% RSLogix 500 project Automated Water Storage & Filtration Control System.RSS, saved by version 8.30.00.16 %
PROJECT "UNTITLED"    % processor: Bul.1763 MicroLogix 1100 Series B %

PROGRAM FILES
  LAD 2 "MAIN"  9 rungs
  LAD 3 "IO"  13 rungs
  LAD 4 "HOA"  36 rungs
  LAD 5 "CONTROLS"  16 rungs
  LAD 6 "RUNTIME"  6 rungs
  LAD 7 "BACKWASH"  16 rungs
  LAD 8 "ALARM"  17 rungs
  LAD 9 "SIMULATION"  9 rungs  % SIMULATED IO %
  LAD 10 "SETTOAUTO"  3 rungs

DATA FILES
  O0 OUTPUT  4 elements
  I1 INPUT  13 elements
  S2 STATUS  66 elements
  B3 BINARY  9 elements
  T4 TIMER  11 elements
  C5 COUNTER  1 elements
  R6 CONTROL  1 elements
  N7 INTEGER  19 elements
  F8 FLOAT  15 elements

LADDER 2 "MAIN"
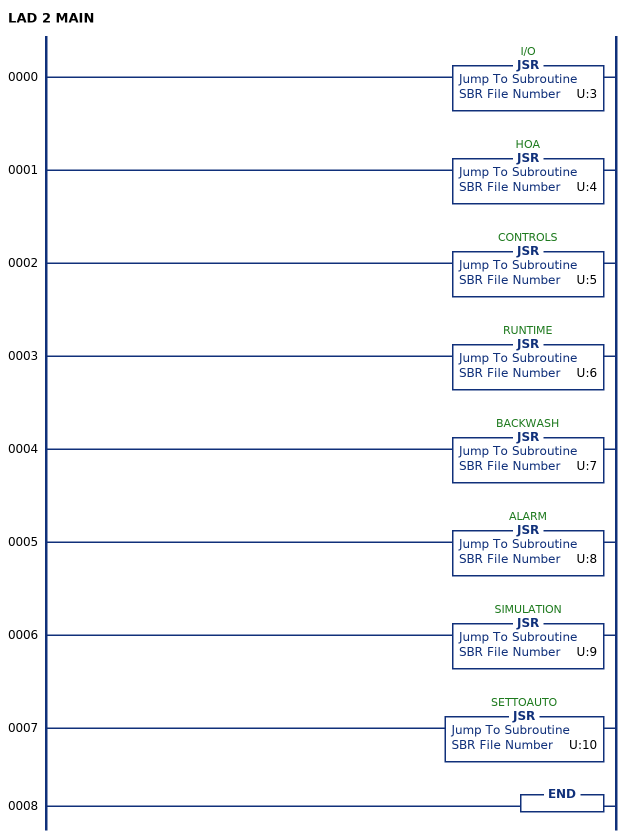
% Rung: 0 %
SOR JSR U:3 EOR
%   U:3  "I/O" %
% Rung: 1 %
SOR JSR U:4 EOR
%   U:4  "HOA" %
% Rung: 2 %
SOR JSR U:5 EOR
%   U:5  "CONTROLS" %
% Rung: 3 %
SOR JSR U:6 EOR
%   U:6  "RUNTIME" %
% Rung: 4 %
SOR JSR U:7 EOR
%   U:7  "BACKWASH" %
% Rung: 5 %
SOR JSR U:8 EOR
%   U:8  "ALARM" %
% Rung: 6 %
SOR JSR U:9 EOR
%   U:9  "SIMULATION" %
% Rung: 7 %
SOR JSR U:10 EOR
%   U:10  "SETTOAUTO" %
% Rung: 8 %
SOR END EOR

LADDER 3 "IO"
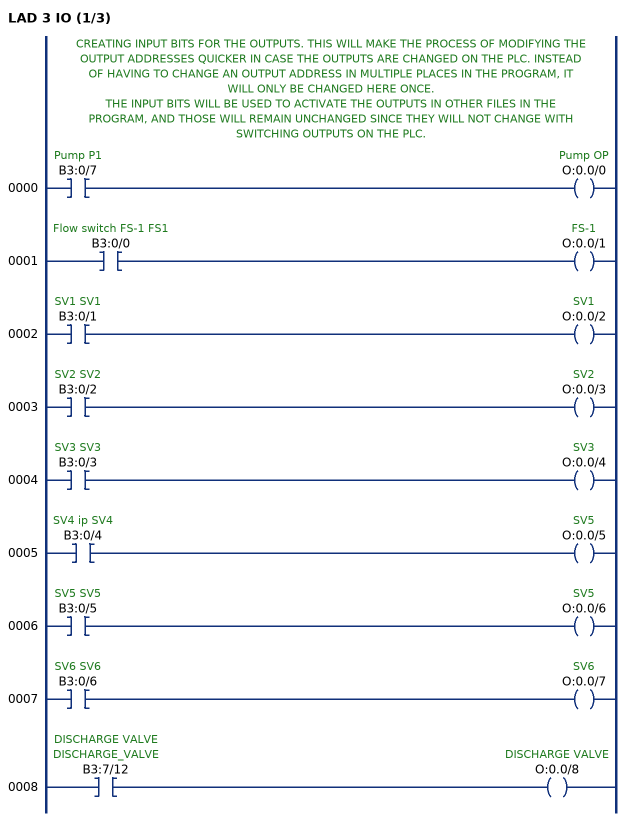
% Rung: 0 %
% CREATING INPUT BITS FOR THE OUTPUTS. THIS WILL MAKE THE PROCESS OF MODIFYING THE OUTPUT ADDRESSES QUICKER IN CASE THE OUTPUTS ARE CHANGED ON THE PLC. INSTEAD OF HAVING TO CHANGE AN OUTPUT ADDRESS IN MULTIPLE PLACES IN THE PROGRAM, IT WILL ONLY BE CHANGED HERE ONCE.
% THE INPUT BITS WILL BE USED TO ACTIVATE THE OUTPUTS IN OTHER FILES IN THE PROGRAM, AND THOSE WILL REMAIN UNCHANGED SINCE THEY WILL NOT CHANGE WITH SWITCHING OUTPUTS ON THE PLC. %
SOR XIC B3:0/7 OTE O:0.0/0 EOR
%   B3:0/7  P1  "Pump" %
%   O:0.0/0  "Pump OP" %
% Rung: 1 %
SOR XIC B3:0/0 OTE O:0.0/1 EOR
%   B3:0/0  FS1  "Flow switch FS-1" %
%   O:0.0/1  "FS-1" %
% Rung: 2 %
SOR XIC B3:0/1 OTE O:0.0/2 EOR
%   B3:0/1  SV1  "SV1" %
%   O:0.0/2  "SV1" %
% Rung: 3 %
SOR XIC B3:0/2 OTE O:0.0/3 EOR
%   B3:0/2  SV2  "SV2" %
%   O:0.0/3  "SV2" %
% Rung: 4 %
SOR XIC B3:0/3 OTE O:0.0/4 EOR
%   B3:0/3  SV3  "SV3" %
%   O:0.0/4  "SV3" %
% Rung: 5 %
SOR XIC B3:0/4 OTE O:0.0/5 EOR
%   B3:0/4  SV4  "SV4 ip" %
%   O:0.0/5  "SV5" %
% Rung: 6 %
SOR XIC B3:0/5 OTE O:0.0/6 EOR
%   B3:0/5  SV5  "SV5" %
%   O:0.0/6  "SV5" %
% Rung: 7 %
SOR XIC B3:0/6 OTE O:0.0/7 EOR
%   B3:0/6  SV6  "SV6" %
%   O:0.0/7  "SV6" %
% Rung: 8 %
SOR XIC B3:7/12 OTE O:0.0/8 EOR
%   B3:7/12  DISCHARGE_VALVE  "DISCHARGE VALVE" %
%   O:0.0/8  "DISCHARGE VALVE" %

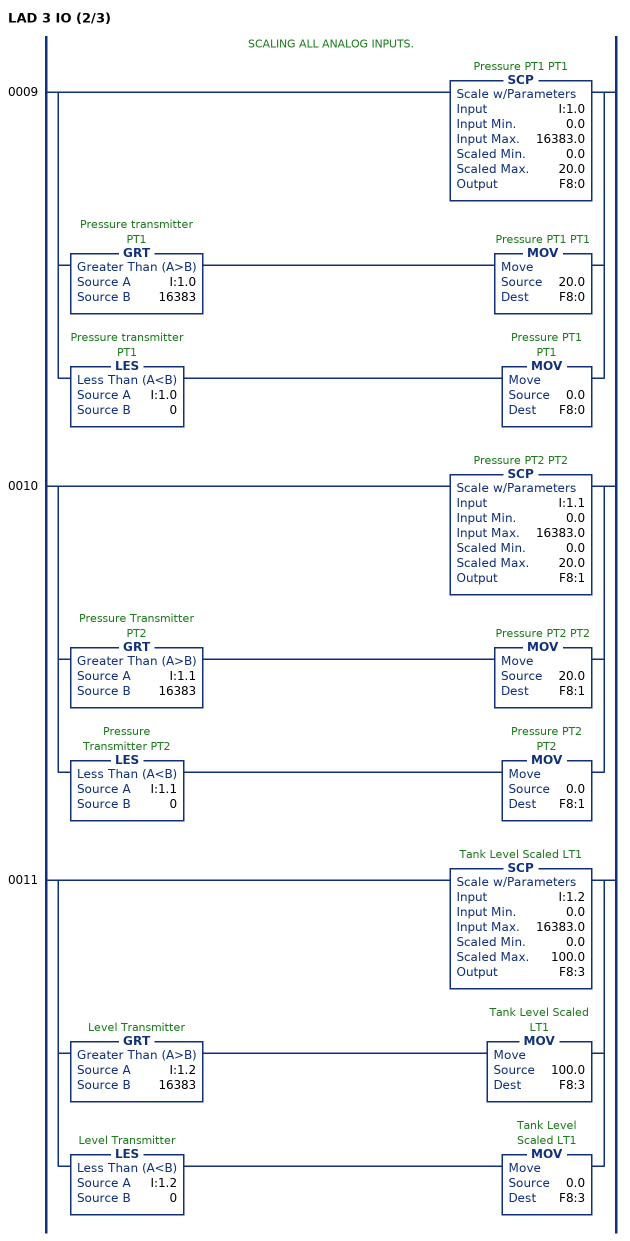
% Rung: 9 %
% SCALING ALL ANALOG INPUTS. %
SOR BST SCP I:1.0 0.0 16383.0 0.0 20.0 F8:0 NXB GRT I:1.0 16383 MOV 20.0 F8:0 NXB LES I:1.0 0 MOV 0.0 F8:0 BND EOR
%   I:1.0  "Pressure transmitter PT1" %
%   F8:0  PT1  "Pressure PT1" %
% Rung: 10 %
SOR BST SCP I:1.1 0.0 16383.0 0.0 20.0 F8:1 NXB GRT I:1.1 16383 MOV 20.0 F8:1 NXB LES I:1.1 0 MOV 0.0 F8:1 BND EOR
%   I:1.1  "Pressure Transmitter PT2" %
%   F8:1  PT2  "Pressure PT2" %
% Rung: 11 %
SOR BST SCP I:1.2 0.0 16383.0 0.0 100.0 F8:3 NXB GRT I:1.2 16383 MOV 100.0 F8:3 NXB LES I:1.2 0 MOV 0.0 F8:3 BND EOR
%   I:1.2  "Level Transmitter" %
%   F8:3  LT1  "Tank Level Scaled" %

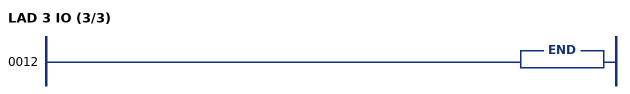
% Rung: 12 %
SOR END EOR

LADDER 4 "HOA"
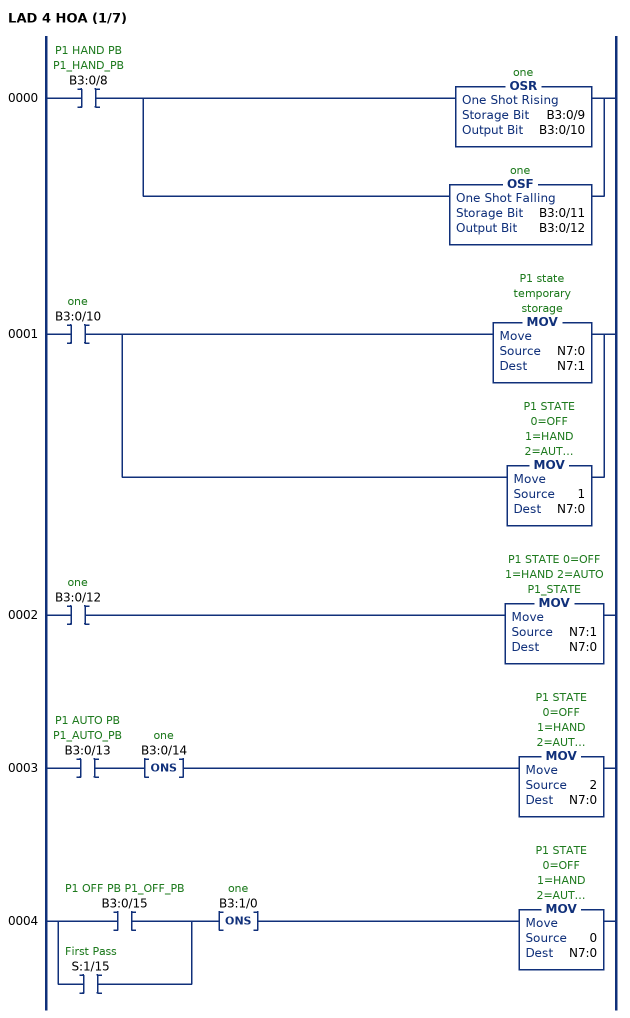
% Rung: 0 %
SOR XIC B3:0/8 BST OSR B3:0/9 B3:0/10 NXB OSF B3:0/11 B3:0/12 BND EOR
%   B3:0/8  P1_HAND_PB  "P1 HAND PB" %
%   B3:0/9  "one" %
%   B3:0/10  "one" %
%   B3:0/11  "one" %
%   B3:0/12  "one" %
% Rung: 1 %
SOR XIC B3:0/10 BST MOV N7:0 N7:1 NXB MOV 1 N7:0 BND EOR
%   B3:0/10  "one" %
%   N7:0  P1_STATE  "P1 STATE 0=OFF 1=HAND 2=AUTO" %
%   N7:1  "P1 state temporary storage" %
% Rung: 2 %
SOR XIC B3:0/12 MOV N7:1 N7:0 EOR
%   B3:0/12  "one" %
%   N7:1  "P1 state temporary storage" %
%   N7:0  P1_STATE  "P1 STATE 0=OFF 1=HAND 2=AUTO" %
% Rung: 3 %
SOR XIC B3:0/13 ONS B3:0/14 MOV 2 N7:0 EOR
%   B3:0/13  P1_AUTO_PB  "P1 AUTO PB" %
%   B3:0/14  "one" %
%   N7:0  P1_STATE  "P1 STATE 0=OFF 1=HAND 2=AUTO" %
% Rung: 4 %
SOR BST XIC B3:0/15 NXB XIC S:1/15 BND ONS B3:1/0 MOV 0 N7:0 EOR
%   B3:0/15  P1_OFF_PB  "P1 OFF PB" %
%   S:1/15  "First Pass" %
%   B3:1/0  "one" %
%   N7:0  P1_STATE  "P1 STATE 0=OFF 1=HAND 2=AUTO" %

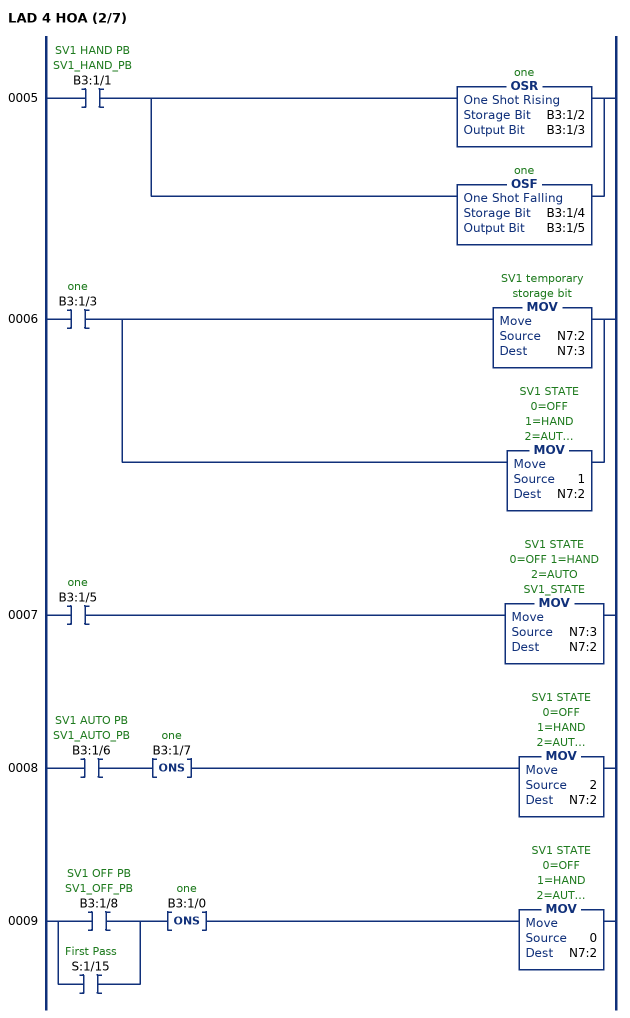
% Rung: 5 %
SOR XIC B3:1/1 BST OSR B3:1/2 B3:1/3 NXB OSF B3:1/4 B3:1/5 BND EOR
%   B3:1/1  SV1_HAND_PB  "SV1 HAND PB" %
%   B3:1/2  "one" %
%   B3:1/3  "one" %
%   B3:1/4  "one" %
%   B3:1/5  "one" %
% Rung: 6 %
SOR XIC B3:1/3 BST MOV N7:2 N7:3 NXB MOV 1 N7:2 BND EOR
%   B3:1/3  "one" %
%   N7:2  SV1_STATE  "SV1 STATE 0=OFF 1=HAND 2=AUTO" %
%   N7:3  "SV1 temporary storage bit" %
% Rung: 7 %
SOR XIC B3:1/5 MOV N7:3 N7:2 EOR
%   B3:1/5  "one" %
%   N7:3  "SV1 temporary storage bit" %
%   N7:2  SV1_STATE  "SV1 STATE 0=OFF 1=HAND 2=AUTO" %
% Rung: 8 %
SOR XIC B3:1/6 ONS B3:1/7 MOV 2 N7:2 EOR
%   B3:1/6  SV1_AUTO_PB  "SV1 AUTO PB" %
%   B3:1/7  "one" %
%   N7:2  SV1_STATE  "SV1 STATE 0=OFF 1=HAND 2=AUTO" %
% Rung: 9 %
SOR BST XIC B3:1/8 NXB XIC S:1/15 BND ONS B3:1/0 MOV 0 N7:2 EOR
%   B3:1/8  SV1_OFF_PB  "SV1 OFF PB" %
%   S:1/15  "First Pass" %
%   B3:1/0  "one" %
%   N7:2  SV1_STATE  "SV1 STATE 0=OFF 1=HAND 2=AUTO" %

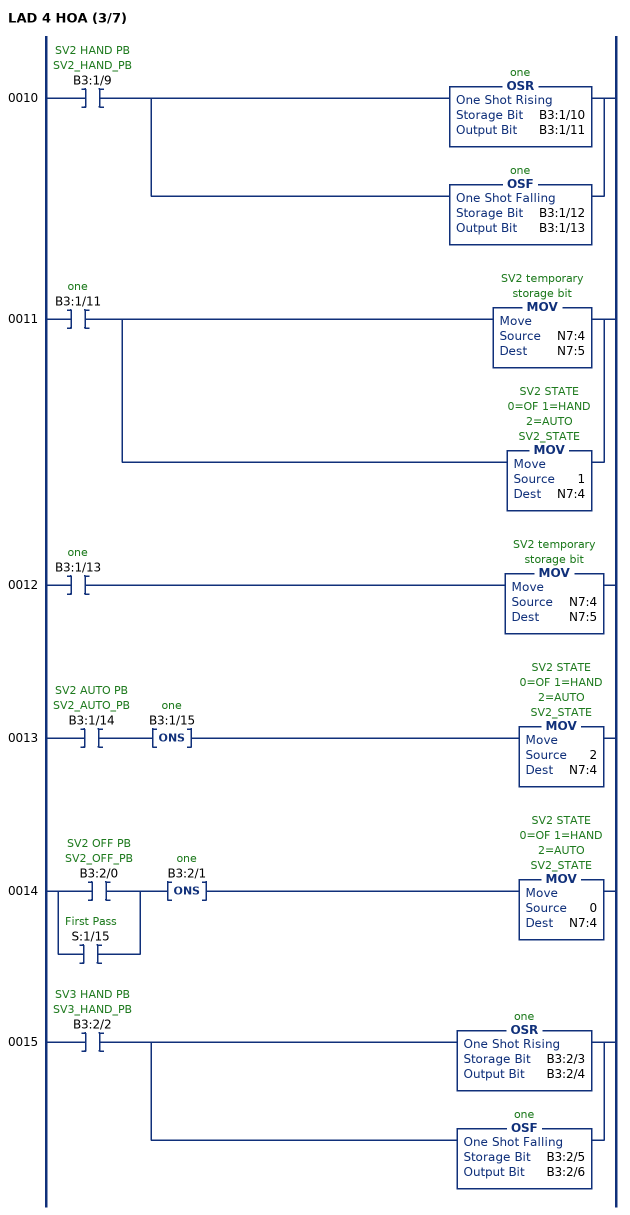
% Rung: 10 %
SOR XIC B3:1/9 BST OSR B3:1/10 B3:1/11 NXB OSF B3:1/12 B3:1/13 BND EOR
%   B3:1/9  SV2_HAND_PB  "SV2 HAND PB" %
%   B3:1/10  "one" %
%   B3:1/11  "one" %
%   B3:1/12  "one" %
%   B3:1/13  "one" %
% Rung: 11 %
SOR XIC B3:1/11 BST MOV N7:4 N7:5 NXB MOV 1 N7:4 BND EOR
%   B3:1/11  "one" %
%   N7:4  SV2_STATE  "SV2 STATE 0=OF 1=HAND 2=AUTO" %
%   N7:5  "SV2 temporary storage bit" %
% Rung: 12 %
SOR XIC B3:1/13 MOV N7:4 N7:5 EOR
%   B3:1/13  "one" %
%   N7:4  SV2_STATE  "SV2 STATE 0=OF 1=HAND 2=AUTO" %
%   N7:5  "SV2 temporary storage bit" %
% Rung: 13 %
SOR XIC B3:1/14 ONS B3:1/15 MOV 2 N7:4 EOR
%   B3:1/14  SV2_AUTO_PB  "SV2 AUTO PB" %
%   B3:1/15  "one" %
%   N7:4  SV2_STATE  "SV2 STATE 0=OF 1=HAND 2=AUTO" %
% Rung: 14 %
SOR BST XIC B3:2/0 NXB XIC S:1/15 BND ONS B3:2/1 MOV 0 N7:4 EOR
%   B3:2/0  SV2_OFF_PB  "SV2 OFF PB" %
%   S:1/15  "First Pass" %
%   B3:2/1  "one" %
%   N7:4  SV2_STATE  "SV2 STATE 0=OF 1=HAND 2=AUTO" %
% Rung: 15 %
SOR XIC B3:2/2 BST OSR B3:2/3 B3:2/4 NXB OSF B3:2/5 B3:2/6 BND EOR
%   B3:2/2  SV3_HAND_PB  "SV3 HAND PB" %
%   B3:2/3  "one" %
%   B3:2/4  "one" %
%   B3:2/5  "one" %
%   B3:2/6  "one" %

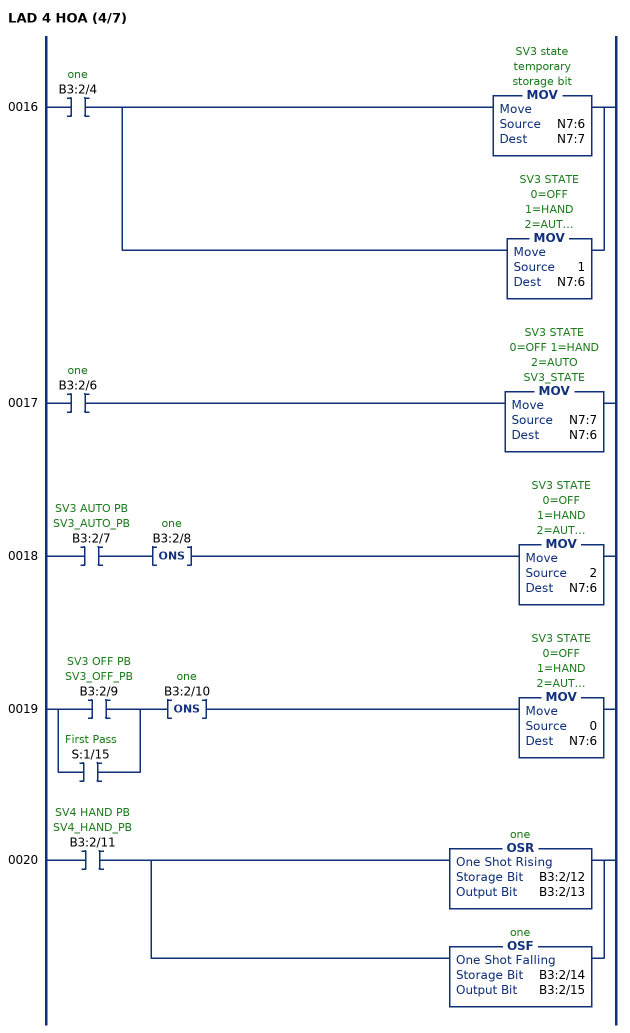
% Rung: 16 %
SOR XIC B3:2/4 BST MOV N7:6 N7:7 NXB MOV 1 N7:6 BND EOR
%   B3:2/4  "one" %
%   N7:6  SV3_STATE  "SV3 STATE 0=OFF 1=HAND 2=AUTO" %
%   N7:7  "SV3 state temporary storage bit" %
% Rung: 17 %
SOR XIC B3:2/6 MOV N7:7 N7:6 EOR
%   B3:2/6  "one" %
%   N7:7  "SV3 state temporary storage bit" %
%   N7:6  SV3_STATE  "SV3 STATE 0=OFF 1=HAND 2=AUTO" %
% Rung: 18 %
SOR XIC B3:2/7 ONS B3:2/8 MOV 2 N7:6 EOR
%   B3:2/7  SV3_AUTO_PB  "SV3 AUTO PB" %
%   B3:2/8  "one" %
%   N7:6  SV3_STATE  "SV3 STATE 0=OFF 1=HAND 2=AUTO" %
% Rung: 19 %
SOR BST XIC B3:2/9 NXB XIC S:1/15 BND ONS B3:2/10 MOV 0 N7:6 EOR
%   B3:2/9  SV3_OFF_PB  "SV3 OFF PB" %
%   S:1/15  "First Pass" %
%   B3:2/10  "one" %
%   N7:6  SV3_STATE  "SV3 STATE 0=OFF 1=HAND 2=AUTO" %
% Rung: 20 %
SOR XIC B3:2/11 BST OSR B3:2/12 B3:2/13 NXB OSF B3:2/14 B3:2/15 BND EOR
%   B3:2/11  SV4_HAND_PB  "SV4 HAND PB" %
%   B3:2/12  "one" %
%   B3:2/13  "one" %
%   B3:2/14  "one" %
%   B3:2/15  "one" %

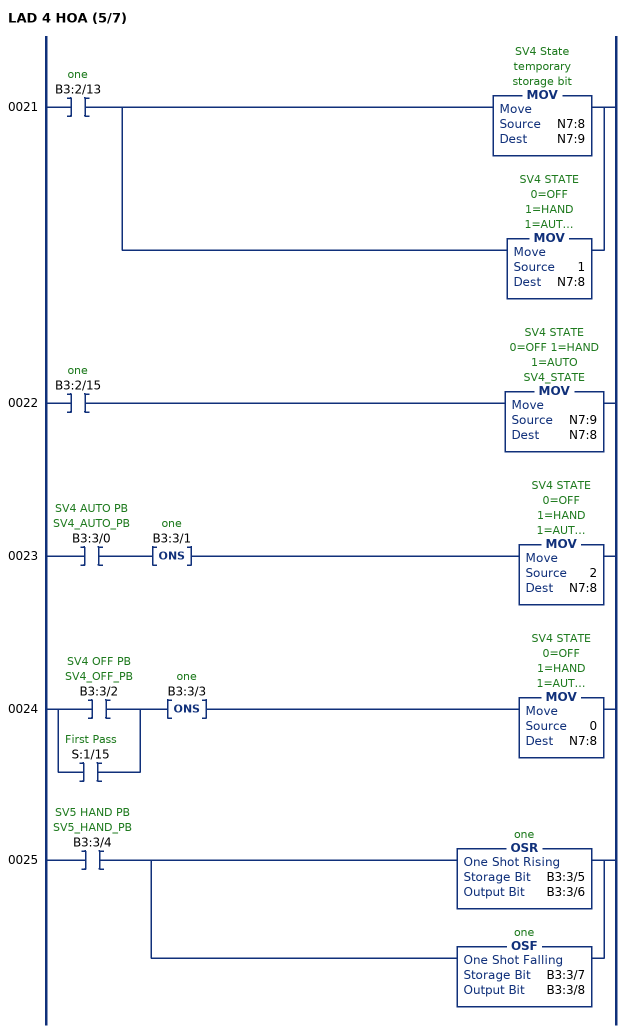
% Rung: 21 %
SOR XIC B3:2/13 BST MOV N7:8 N7:9 NXB MOV 1 N7:8 BND EOR
%   B3:2/13  "one" %
%   N7:8  SV4_STATE  "SV4 STATE 0=OFF 1=HAND 1=AUTO" %
%   N7:9  "SV4 State temporary storage bit" %
% Rung: 22 %
SOR XIC B3:2/15 MOV N7:9 N7:8 EOR
%   B3:2/15  "one" %
%   N7:9  "SV4 State temporary storage bit" %
%   N7:8  SV4_STATE  "SV4 STATE 0=OFF 1=HAND 1=AUTO" %
% Rung: 23 %
SOR XIC B3:3/0 ONS B3:3/1 MOV 2 N7:8 EOR
%   B3:3/0  SV4_AUTO_PB  "SV4 AUTO PB" %
%   B3:3/1  "one" %
%   N7:8  SV4_STATE  "SV4 STATE 0=OFF 1=HAND 1=AUTO" %
% Rung: 24 %
SOR BST XIC B3:3/2 NXB XIC S:1/15 BND ONS B3:3/3 MOV 0 N7:8 EOR
%   B3:3/2  SV4_OFF_PB  "SV4 OFF PB" %
%   S:1/15  "First Pass" %
%   B3:3/3  "one" %
%   N7:8  SV4_STATE  "SV4 STATE 0=OFF 1=HAND 1=AUTO" %
% Rung: 25 %
SOR XIC B3:3/4 BST OSR B3:3/5 B3:3/6 NXB OSF B3:3/7 B3:3/8 BND EOR
%   B3:3/4  SV5_HAND_PB  "SV5 HAND PB" %
%   B3:3/5  "one" %
%   B3:3/6  "one" %
%   B3:3/7  "one" %
%   B3:3/8  "one" %

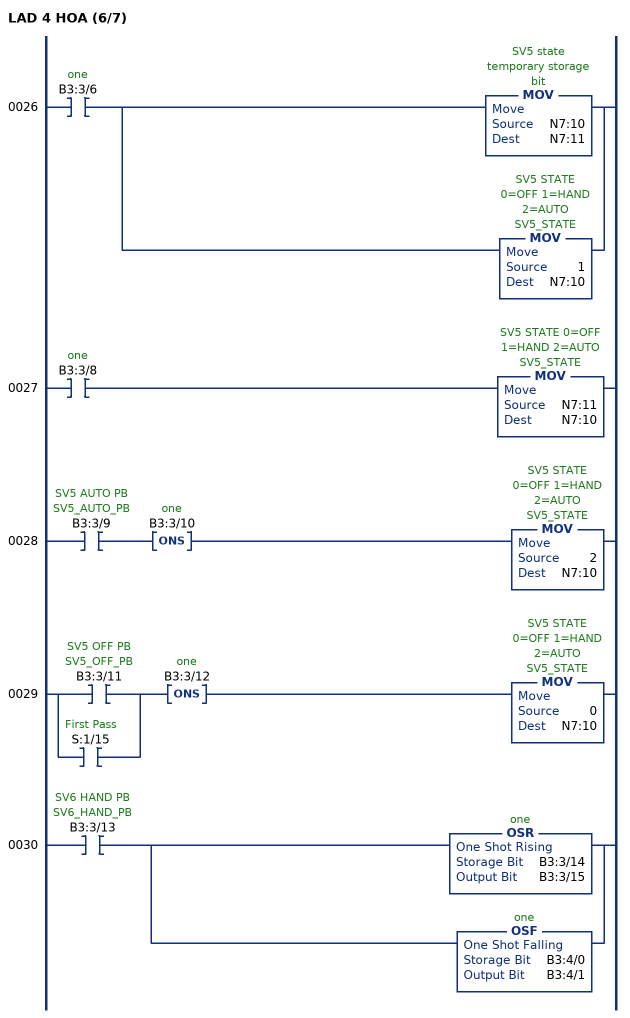
% Rung: 26 %
SOR XIC B3:3/6 BST MOV N7:10 N7:11 NXB MOV 1 N7:10 BND EOR
%   B3:3/6  "one" %
%   N7:10  SV5_STATE  "SV5 STATE 0=OFF 1=HAND 2=AUTO" %
%   N7:11  "SV5 state temporary storage bit" %
% Rung: 27 %
SOR XIC B3:3/8 MOV N7:11 N7:10 EOR
%   B3:3/8  "one" %
%   N7:11  "SV5 state temporary storage bit" %
%   N7:10  SV5_STATE  "SV5 STATE 0=OFF 1=HAND 2=AUTO" %
% Rung: 28 %
SOR XIC B3:3/9 ONS B3:3/10 MOV 2 N7:10 EOR
%   B3:3/9  SV5_AUTO_PB  "SV5 AUTO PB" %
%   B3:3/10  "one" %
%   N7:10  SV5_STATE  "SV5 STATE 0=OFF 1=HAND 2=AUTO" %
% Rung: 29 %
SOR BST XIC B3:3/11 NXB XIC S:1/15 BND ONS B3:3/12 MOV 0 N7:10 EOR
%   B3:3/11  SV5_OFF_PB  "SV5 OFF PB" %
%   S:1/15  "First Pass" %
%   B3:3/12  "one" %
%   N7:10  SV5_STATE  "SV5 STATE 0=OFF 1=HAND 2=AUTO" %
% Rung: 30 %
SOR XIC B3:3/13 BST OSR B3:3/14 B3:3/15 NXB OSF B3:4/0 B3:4/1 BND EOR
%   B3:3/13  SV6_HAND_PB  "SV6 HAND PB" %
%   B3:3/14  "one" %
%   B3:3/15  "one" %
%   B3:4/0  "one" %
%   B3:4/1  "one" %

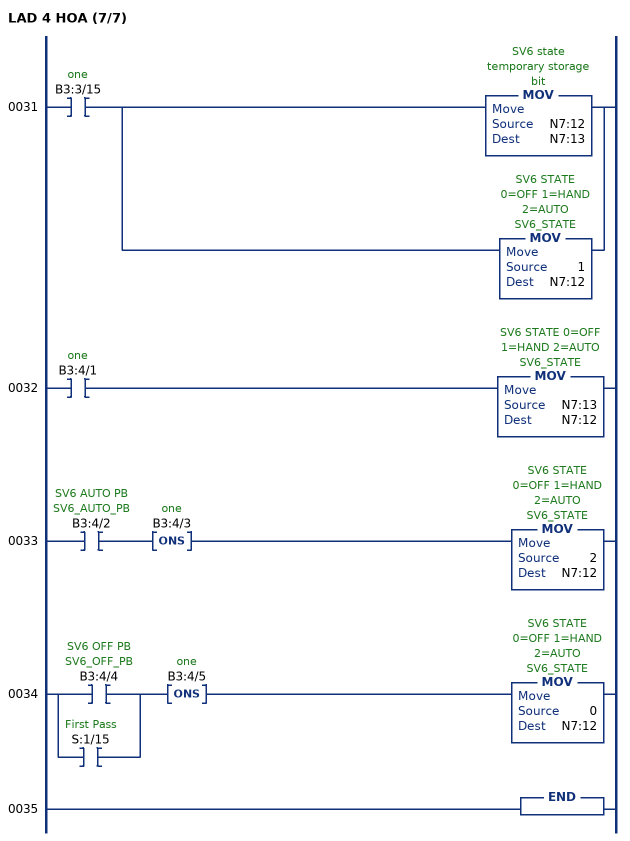
% Rung: 31 %
SOR XIC B3:3/15 BST MOV N7:12 N7:13 NXB MOV 1 N7:12 BND EOR
%   B3:3/15  "one" %
%   N7:12  SV6_STATE  "SV6 STATE 0=OFF 1=HAND 2=AUTO" %
%   N7:13  "SV6 state temporary storage bit" %
% Rung: 32 %
SOR XIC B3:4/1 MOV N7:13 N7:12 EOR
%   B3:4/1  "one" %
%   N7:13  "SV6 state temporary storage bit" %
%   N7:12  SV6_STATE  "SV6 STATE 0=OFF 1=HAND 2=AUTO" %
% Rung: 33 %
SOR XIC B3:4/2 ONS B3:4/3 MOV 2 N7:12 EOR
%   B3:4/2  SV6_AUTO_PB  "SV6 AUTO PB" %
%   B3:4/3  "one" %
%   N7:12  SV6_STATE  "SV6 STATE 0=OFF 1=HAND 2=AUTO" %
% Rung: 34 %
SOR BST XIC B3:4/4 NXB XIC S:1/15 BND ONS B3:4/5 MOV 0 N7:12 EOR
%   B3:4/4  SV6_OFF_PB  "SV6 OFF PB" %
%   S:1/15  "First Pass" %
%   B3:4/5  "one" %
%   N7:12  SV6_STATE  "SV6 STATE 0=OFF 1=HAND 2=AUTO" %
% Rung: 35 %
SOR END EOR

LADDER 5 "CONTROLS"
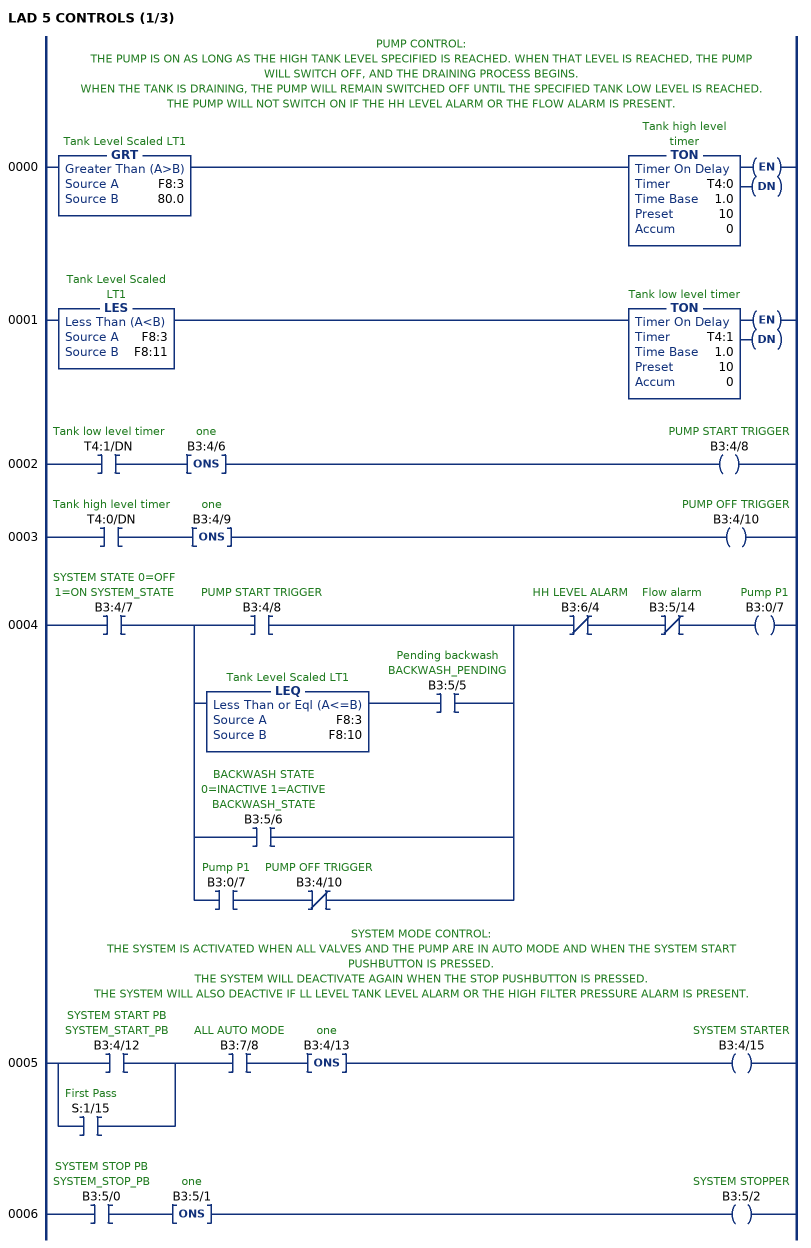
% Rung: 0 %
% PUMP CONTROL:
% THE PUMP IS ON AS LONG AS THE HIGH TANK LEVEL SPECIFIED IS REACHED. WHEN THAT LEVEL IS REACHED, THE PUMP WILL SWITCH OFF, AND THE DRAINING PROCESS BEGINS.
% WHEN THE TANK IS DRAINING, THE PUMP WILL REMAIN SWITCHED OFF UNTIL THE SPECIFIED TANK LOW LEVEL IS REACHED.
% THE PUMP WILL NOT SWITCH ON IF THE HH LEVEL ALARM OR THE FLOW ALARM IS PRESENT. %
SOR GRT F8:3 80.0 TON T4:0 1.0 10 0 EOR
%   F8:3  LT1  "Tank Level Scaled" %
%   T4:0  "Tank high level timer" %
% Rung: 1 %
SOR LES F8:3 F8:11 TON T4:1 1.0 10 0 EOR
%   F8:3  LT1  "Tank Level Scaled" %
%   F8:11  L_LEVEL  "L_TANK_LEVEL" %
%   T4:1  "Tank low level timer" %
% Rung: 2 %
SOR XIC T4:1/DN ONS B3:4/6 OTE B3:4/8 EOR
%   T4:1  "Tank low level timer" %
%   B3:4/6  "one" %
%   B3:4/8  "PUMP START TRIGGER" %
% Rung: 3 %
SOR XIC T4:0/DN ONS B3:4/9 OTE B3:4/10 EOR
%   T4:0  "Tank high level timer" %
%   B3:4/9  "one" %
%   B3:4/10  "PUMP OFF TRIGGER" %
% Rung: 4 %
SOR XIC B3:4/7 BST XIC B3:4/8 NXB LEQ F8:3 F8:10 XIC B3:5/5 NXB XIC B3:5/6 NXB XIC B3:0/7 XIO B3:4/10 BND XIO B3:6/4 XIO B3:5/14 OTE B3:0/7 EOR
%   B3:4/7  SYSTEM_STATE  "SYSTEM STATE 0=OFF 1=ON" %
%   B3:4/8  "PUMP START TRIGGER" %
%   F8:3  LT1  "Tank Level Scaled" %
%   F8:10  H_LEVEL  "H_TANK_LEVEL" %
%   B3:5/5  BACKWASH_PENDING  "Pending backwash" %
%   B3:5/6  BACKWASH_STATE  "BACKWASH STATE 0=INACTIVE 1=ACTIVE" %
%   B3:0/7  P1  "Pump" %
%   B3:4/10  "PUMP OFF TRIGGER" %
%   B3:6/4  "HH LEVEL ALARM" %
%   B3:5/14  "Flow alarm" %
% Rung: 5 %
% SYSTEM MODE CONTROL:
% THE SYSTEM IS ACTIVATED WHEN ALL VALVES AND THE PUMP ARE IN AUTO MODE AND WHEN THE SYSTEM START PUSHBUTTON IS PRESSED.
% THE SYSTEM WILL DEACTIVATE AGAIN WHEN THE STOP PUSHBUTTON IS PRESSED.
% THE SYSTEM WILL ALSO DEACTIVE IF LL LEVEL TANK LEVEL ALARM OR THE HIGH FILTER PRESSURE ALARM IS PRESENT. %
SOR BST XIC B3:4/12 NXB XIC S:1/15 BND XIC B3:7/8 ONS B3:4/13 OTE B3:4/15 EOR
%   B3:4/12  SYSTEM_START_PB  "SYSTEM START PB" %
%   S:1/15  "First Pass" %
%   B3:7/8  "ALL AUTO MODE" %
%   B3:4/13  "one" %
%   B3:4/15  "SYSTEM STARTER" %
% Rung: 6 %
SOR XIC B3:5/0 ONS B3:5/1 OTE B3:5/2 EOR
%   B3:5/0  SYSTEM_STOP_PB  "SYSTEM STOP PB" %
%   B3:5/1  "one" %
%   B3:5/2  "SYSTEM STOPPER" %

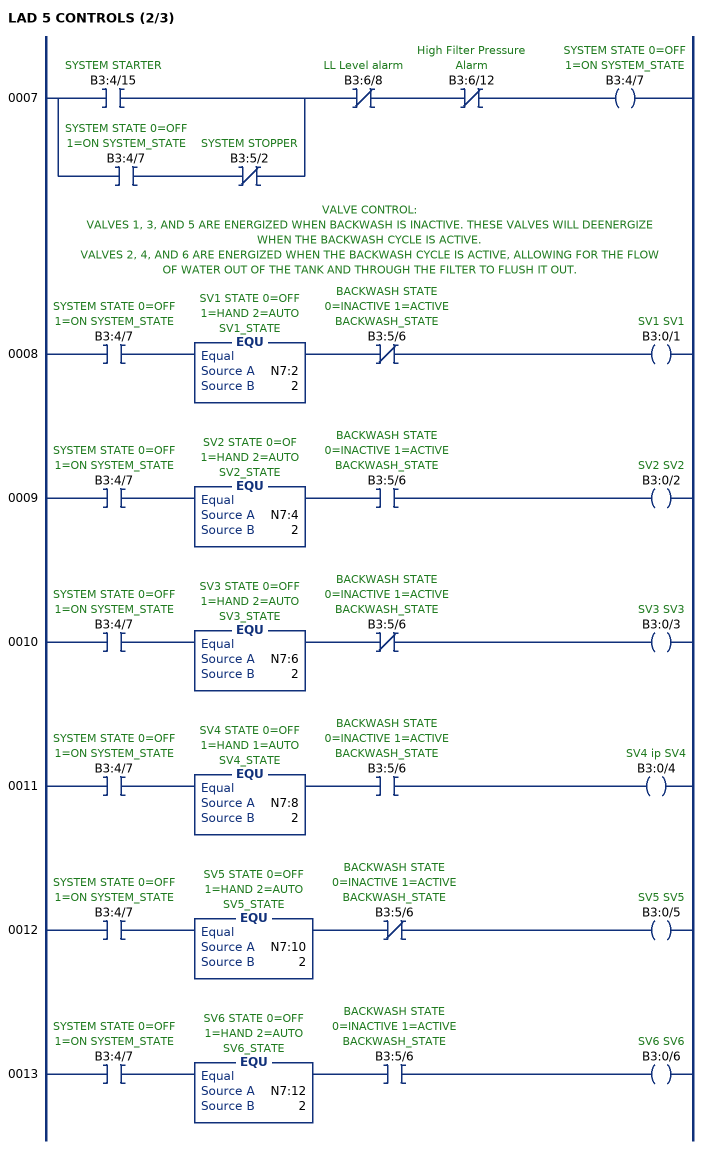
% Rung: 7 %
SOR BST XIC B3:4/15 NXB XIC B3:4/7 XIO B3:5/2 BND XIO B3:6/8 XIO B3:6/12 OTE B3:4/7 EOR
%   B3:4/15  "SYSTEM STARTER" %
%   B3:4/7  SYSTEM_STATE  "SYSTEM STATE 0=OFF 1=ON" %
%   B3:5/2  "SYSTEM STOPPER" %
%   B3:6/8  "LL Level alarm" %
%   B3:6/12  "High Filter Pressure Alarm" %
% Rung: 8 %
% VALVE CONTROL:
% VALVES 1, 3, AND 5 ARE ENERGIZED WHEN BACKWASH IS INACTIVE. THESE VALVES WILL DEENERGIZE WHEN THE BACKWASH CYCLE IS ACTIVE.
% VALVES 2, 4, AND 6 ARE ENERGIZED WHEN THE BACKWASH CYCLE IS ACTIVE, ALLOWING FOR THE FLOW OF WATER OUT OF THE TANK AND THROUGH THE FILTER TO FLUSH IT OUT. %
SOR XIC B3:4/7 EQU N7:2 2 XIO B3:5/6 OTE B3:0/1 EOR
%   B3:4/7  SYSTEM_STATE  "SYSTEM STATE 0=OFF 1=ON" %
%   N7:2  SV1_STATE  "SV1 STATE 0=OFF 1=HAND 2=AUTO" %
%   B3:5/6  BACKWASH_STATE  "BACKWASH STATE 0=INACTIVE 1=ACTIVE" %
%   B3:0/1  SV1  "SV1" %
% Rung: 9 %
SOR XIC B3:4/7 EQU N7:4 2 XIC B3:5/6 OTE B3:0/2 EOR
%   B3:4/7  SYSTEM_STATE  "SYSTEM STATE 0=OFF 1=ON" %
%   N7:4  SV2_STATE  "SV2 STATE 0=OF 1=HAND 2=AUTO" %
%   B3:5/6  BACKWASH_STATE  "BACKWASH STATE 0=INACTIVE 1=ACTIVE" %
%   B3:0/2  SV2  "SV2" %
% Rung: 10 %
SOR XIC B3:4/7 EQU N7:6 2 XIO B3:5/6 OTE B3:0/3 EOR
%   B3:4/7  SYSTEM_STATE  "SYSTEM STATE 0=OFF 1=ON" %
%   N7:6  SV3_STATE  "SV3 STATE 0=OFF 1=HAND 2=AUTO" %
%   B3:5/6  BACKWASH_STATE  "BACKWASH STATE 0=INACTIVE 1=ACTIVE" %
%   B3:0/3  SV3  "SV3" %
% Rung: 11 %
SOR XIC B3:4/7 EQU N7:8 2 XIC B3:5/6 OTE B3:0/4 EOR
%   B3:4/7  SYSTEM_STATE  "SYSTEM STATE 0=OFF 1=ON" %
%   N7:8  SV4_STATE  "SV4 STATE 0=OFF 1=HAND 1=AUTO" %
%   B3:5/6  BACKWASH_STATE  "BACKWASH STATE 0=INACTIVE 1=ACTIVE" %
%   B3:0/4  SV4  "SV4 ip" %
% Rung: 12 %
SOR XIC B3:4/7 EQU N7:10 2 XIO B3:5/6 OTE B3:0/5 EOR
%   B3:4/7  SYSTEM_STATE  "SYSTEM STATE 0=OFF 1=ON" %
%   N7:10  SV5_STATE  "SV5 STATE 0=OFF 1=HAND 2=AUTO" %
%   B3:5/6  BACKWASH_STATE  "BACKWASH STATE 0=INACTIVE 1=ACTIVE" %
%   B3:0/5  SV5  "SV5" %
% Rung: 13 %
SOR XIC B3:4/7 EQU N7:12 2 XIC B3:5/6 OTE B3:0/6 EOR
%   B3:4/7  SYSTEM_STATE  "SYSTEM STATE 0=OFF 1=ON" %
%   N7:12  SV6_STATE  "SV6 STATE 0=OFF 1=HAND 2=AUTO" %
%   B3:5/6  BACKWASH_STATE  "BACKWASH STATE 0=INACTIVE 1=ACTIVE" %
%   B3:0/6  SV6  "SV6" %

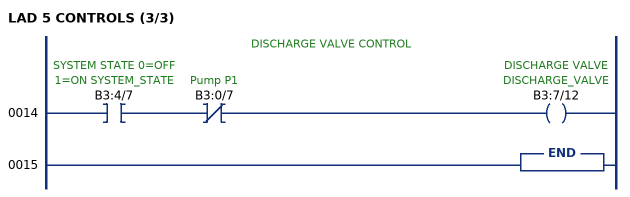
% Rung: 14 %
% DISCHARGE VALVE CONTROL %
SOR XIC B3:4/7 XIO B3:0/7 OTE B3:7/12 EOR
%   B3:4/7  SYSTEM_STATE  "SYSTEM STATE 0=OFF 1=ON" %
%   B3:0/7  P1  "Pump" %
%   B3:7/12  DISCHARGE_VALVE  "DISCHARGE VALVE" %
% Rung: 15 %
SOR END EOR

LADDER 6 "RUNTIME"
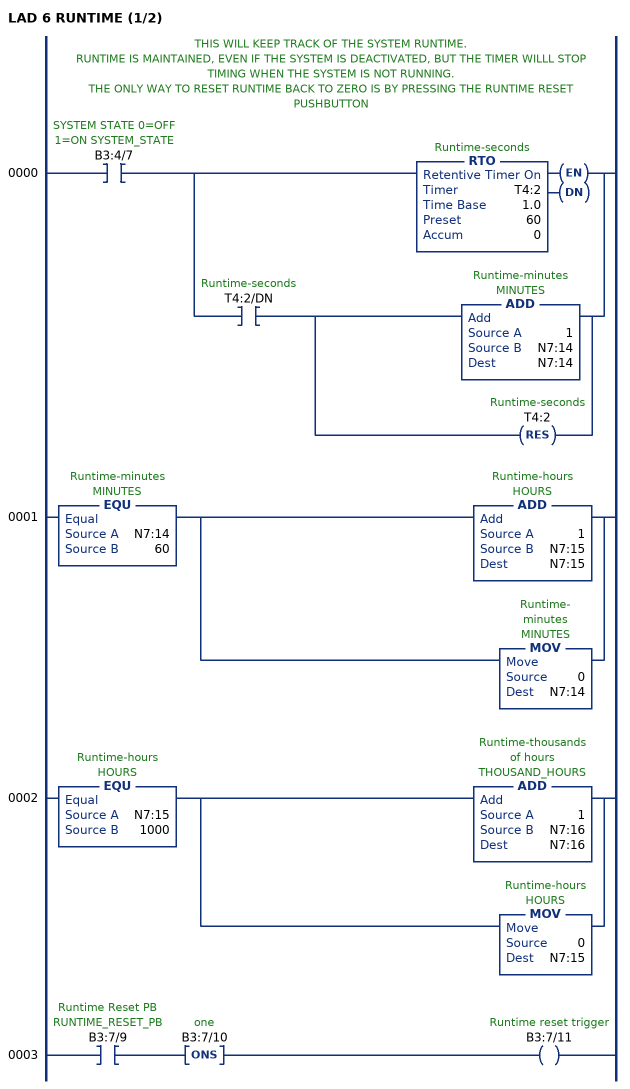
% Rung: 0 %
% THIS WILL KEEP TRACK OF THE SYSTEM RUNTIME.
% RUNTIME IS MAINTAINED, EVEN IF THE SYSTEM IS DEACTIVATED, BUT THE TIMER WILLL STOP TIMING WHEN THE SYSTEM IS NOT RUNNING.
% THE ONLY WAY TO RESET RUNTIME BACK TO ZERO IS BY PRESSING THE RUNTIME RESET PUSHBUTTON %
SOR XIC B3:4/7 BST RTO T4:2 1.0 60 0 NXB XIC T4:2/DN BST ADD 1 N7:14 N7:14 NXB RES T4:2 BND BND EOR
%   B3:4/7  SYSTEM_STATE  "SYSTEM STATE 0=OFF 1=ON" %
%   T4:2  "Runtime-seconds" %
%   N7:14  MINUTES  "Runtime-minutes" %
% Rung: 1 %
SOR EQU N7:14 60 BST ADD 1 N7:15 N7:15 NXB MOV 0 N7:14 BND EOR
%   N7:14  MINUTES  "Runtime-minutes" %
%   N7:15  HOURS  "Runtime-hours" %
% Rung: 2 %
SOR EQU N7:15 1000 BST ADD 1 N7:16 N7:16 NXB MOV 0 N7:15 BND EOR
%   N7:15  HOURS  "Runtime-hours" %
%   N7:16  THOUSAND_HOURS  "Runtime-thousands of hours" %
% Rung: 3 %
SOR XIC B3:7/9 ONS B3:7/10 OTE B3:7/11 EOR
%   B3:7/9  RUNTIME_RESET_PB  "Runtime Reset PB" %
%   B3:7/10  "one" %
%   B3:7/11  "Runtime reset trigger" %

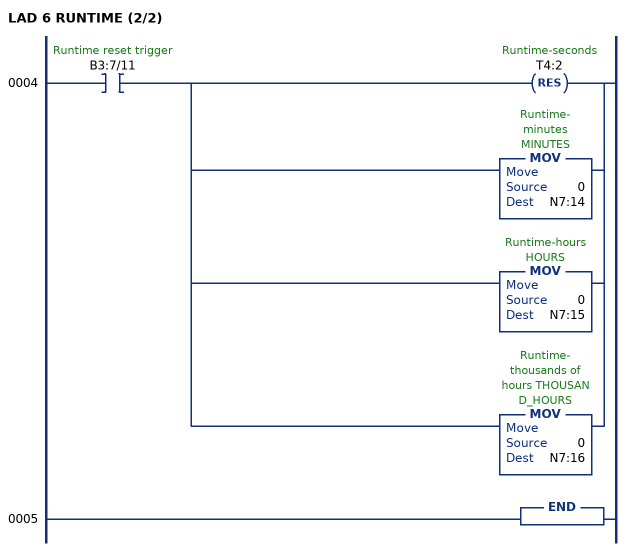
% Rung: 4 %
SOR XIC B3:7/11 BST RES T4:2 NXB MOV 0 N7:14 NXB MOV 0 N7:15 NXB MOV 0 N7:16 BND EOR
%   B3:7/11  "Runtime reset trigger" %
%   T4:2  "Runtime-seconds" %
%   N7:14  MINUTES  "Runtime-minutes" %
%   N7:15  HOURS  "Runtime-hours" %
%   N7:16  THOUSAND_HOURS  "Runtime-thousands of hours" %
% Rung: 5 %
SOR END EOR

LADDER 7 "BACKWASH"
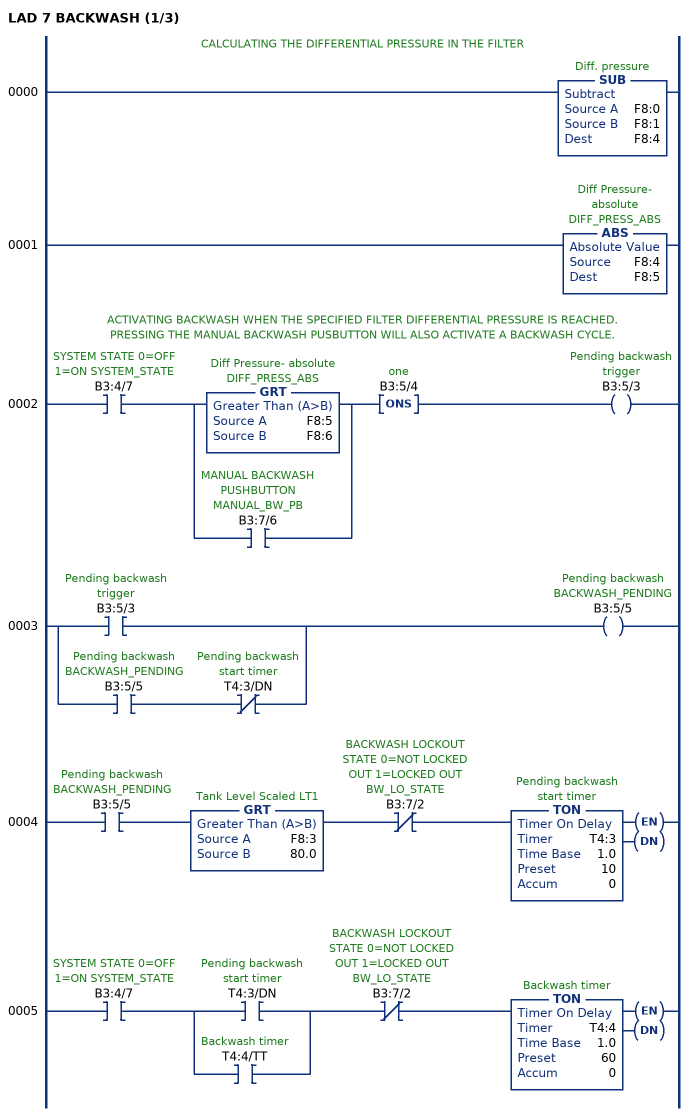
% Rung: 0 %
% CALCULATING THE DIFFERENTIAL PRESSURE IN THE FILTER %
SOR SUB F8:0 F8:1 F8:4 EOR
%   F8:0  PT1  "Pressure PT1" %
%   F8:1  PT2  "Pressure PT2" %
%   F8:4  "Diff. pressure" %
% Rung: 1 %
SOR ABS F8:4 F8:5 EOR
%   F8:4  "Diff. pressure" %
%   F8:5  DIFF_PRESS_ABS  "Diff Pressure- absolute" %
% Rung: 2 %
% ACTIVATING BACKWASH WHEN THE SPECIFIED FILTER DIFFERENTIAL PRESSURE IS REACHED.
% PRESSING THE MANUAL BACKWASH PUSBUTTON WILL ALSO ACTIVATE A BACKWASH CYCLE. %
SOR XIC B3:4/7 BST GRT F8:5 F8:6 NXB XIC B3:7/6 BND ONS B3:5/4 OTE B3:5/3 EOR
%   B3:4/7  SYSTEM_STATE  "SYSTEM STATE 0=OFF 1=ON" %
%   F8:5  DIFF_PRESS_ABS  "Diff Pressure- absolute" %
%   F8:6  DIFF_PRES_SP  "Max. Diff Pressue (set from HMI)" %
%   B3:7/6  MANUAL_BW_PB  "MANUAL BACKWASH PUSHBUTTON" %
%   B3:5/4  "one" %
%   B3:5/3  "Pending backwash trigger" %
% Rung: 3 %
SOR BST XIC B3:5/3 NXB XIC B3:5/5 XIO T4:3/DN BND OTE B3:5/5 EOR
%   B3:5/3  "Pending backwash trigger" %
%   B3:5/5  BACKWASH_PENDING  "Pending backwash" %
%   T4:3  "Pending backwash start timer" %
% Rung: 4 %
SOR XIC B3:5/5 GRT F8:3 80.0 XIO B3:7/2 TON T4:3 1.0 10 0 EOR
%   B3:5/5  BACKWASH_PENDING  "Pending backwash" %
%   F8:3  LT1  "Tank Level Scaled" %
%   B3:7/2  BW_LO_STATE  "BACKWASH LOCKOUT STATE 0=NOT LOCKED OUT 1=LOCKED OUT" %
%   T4:3  "Pending backwash start timer" %
% Rung: 5 %
SOR XIC B3:4/7 BST XIC T4:3/DN NXB XIC T4:4/TT BND XIO B3:7/2 TON T4:4 1.0 60 0 EOR
%   B3:4/7  SYSTEM_STATE  "SYSTEM STATE 0=OFF 1=ON" %
%   T4:3  "Pending backwash start timer" %
%   T4:4  "Backwash timer" %
%   B3:7/2  BW_LO_STATE  "BACKWASH LOCKOUT STATE 0=NOT LOCKED OUT 1=LOCKED OUT" %

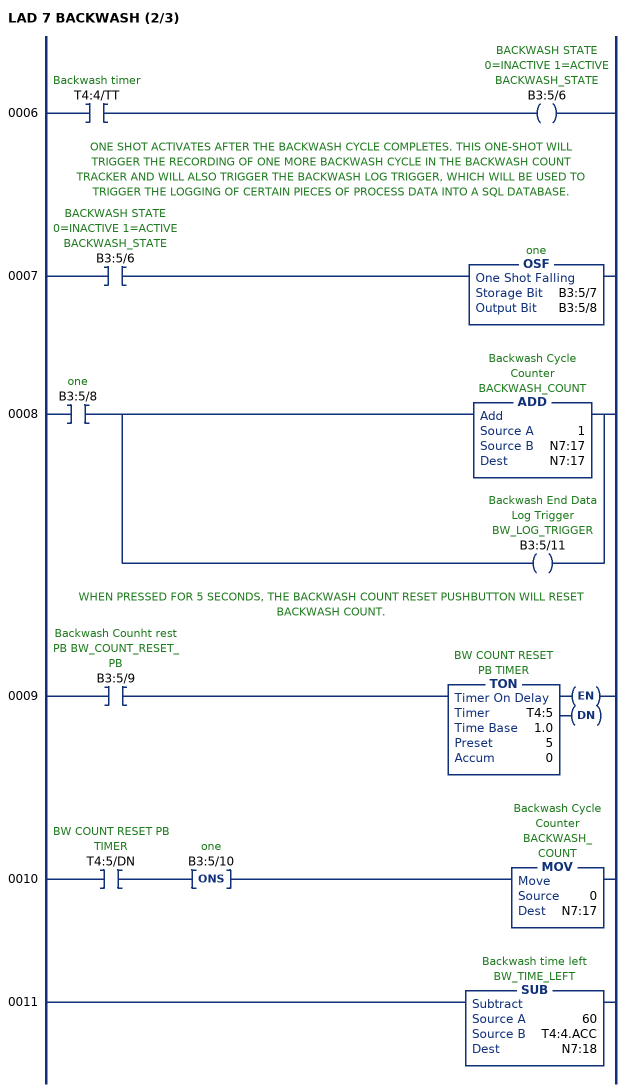
% Rung: 6 %
SOR XIC T4:4/TT OTE B3:5/6 EOR
%   T4:4  "Backwash timer" %
%   B3:5/6  BACKWASH_STATE  "BACKWASH STATE 0=INACTIVE 1=ACTIVE" %
% Rung: 7 %
% ONE SHOT ACTIVATES AFTER THE BACKWASH CYCLE COMPLETES. THIS ONE-SHOT WILL TRIGGER THE RECORDING OF ONE MORE BACKWASH CYCLE IN THE BACKWASH COUNT TRACKER AND WILL ALSO TRIGGER THE BACKWASH LOG TRIGGER, WHICH WILL BE USED TO TRIGGER THE LOGGING OF CERTAIN PIECES OF PROCESS DATA INTO A SQL DATABASE. %
SOR XIC B3:5/6 OSF B3:5/7 B3:5/8 EOR
%   B3:5/6  BACKWASH_STATE  "BACKWASH STATE 0=INACTIVE 1=ACTIVE" %
%   B3:5/7  "one" %
%   B3:5/8  "one" %
% Rung: 8 %
SOR XIC B3:5/8 BST ADD 1 N7:17 N7:17 NXB OTE B3:5/11 BND EOR
%   B3:5/8  "one" %
%   N7:17  BACKWASH_COUNT  "Backwash Cycle Counter" %
%   B3:5/11  BW_LOG_TRIGGER  "Backwash End Data Log Trigger" %
% Rung: 9 %
% WHEN PRESSED FOR 5 SECONDS, THE BACKWASH COUNT RESET PUSHBUTTON WILL RESET BACKWASH COUNT. %
SOR XIC B3:5/9 TON T4:5 1.0 5 0 EOR
%   B3:5/9  BW_COUNT_RESET_PB  "Backwash Counht rest PB" %
%   T4:5  "BW COUNT RESET PB TIMER" %
% Rung: 10 %
SOR XIC T4:5/DN ONS B3:5/10 MOV 0 N7:17 EOR
%   T4:5  "BW COUNT RESET PB TIMER" %
%   B3:5/10  "one" %
%   N7:17  BACKWASH_COUNT  "Backwash Cycle Counter" %
% Rung: 11 %
SOR SUB 60 T4:4.ACC N7:18 EOR
%   T4:4  "Backwash timer" %
%   N7:18  BW_TIME_LEFT  "Backwash time left" %

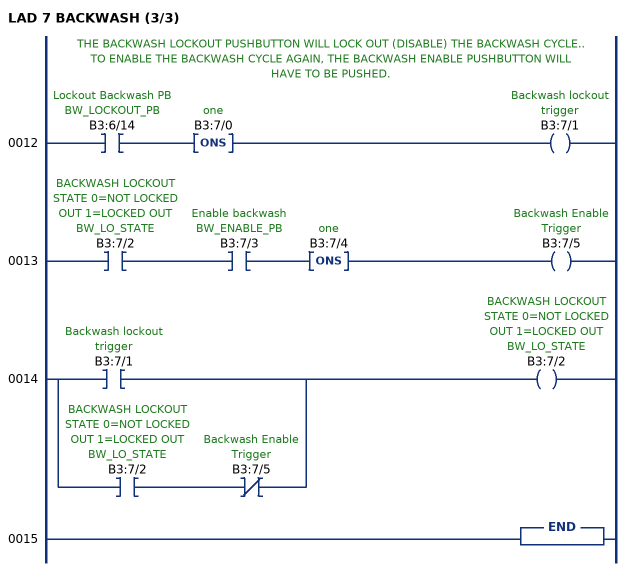
% Rung: 12 %
% THE BACKWASH LOCKOUT PUSHBUTTON WILL LOCK OUT (DISABLE) THE BACKWASH CYCLE..
% TO ENABLE THE BACKWASH CYCLE AGAIN, THE BACKWASH ENABLE PUSHBUTTON WILL HAVE TO BE PUSHED. %
SOR XIC B3:6/14 ONS B3:7/0 OTE B3:7/1 EOR
%   B3:6/14  BW_LOCKOUT_PB  "Lockout Backwash PB" %
%   B3:7/0  "one" %
%   B3:7/1  "Backwash lockout trigger" %
% Rung: 13 %
SOR XIC B3:7/2 XIC B3:7/3 ONS B3:7/4 OTE B3:7/5 EOR
%   B3:7/2  BW_LO_STATE  "BACKWASH LOCKOUT STATE 0=NOT LOCKED OUT 1=LOCKED OUT" %
%   B3:7/3  BW_ENABLE_PB  "Enable backwash" %
%   B3:7/4  "one" %
%   B3:7/5  "Backwash Enable Trigger" %
% Rung: 14 %
SOR BST XIC B3:7/1 NXB XIC B3:7/2 XIO B3:7/5 BND OTE B3:7/2 EOR
%   B3:7/1  "Backwash lockout trigger" %
%   B3:7/2  BW_LO_STATE  "BACKWASH LOCKOUT STATE 0=NOT LOCKED OUT 1=LOCKED OUT" %
%   B3:7/5  "Backwash Enable Trigger" %
% Rung: 15 %
SOR END EOR

LADDER 8 "ALARM"
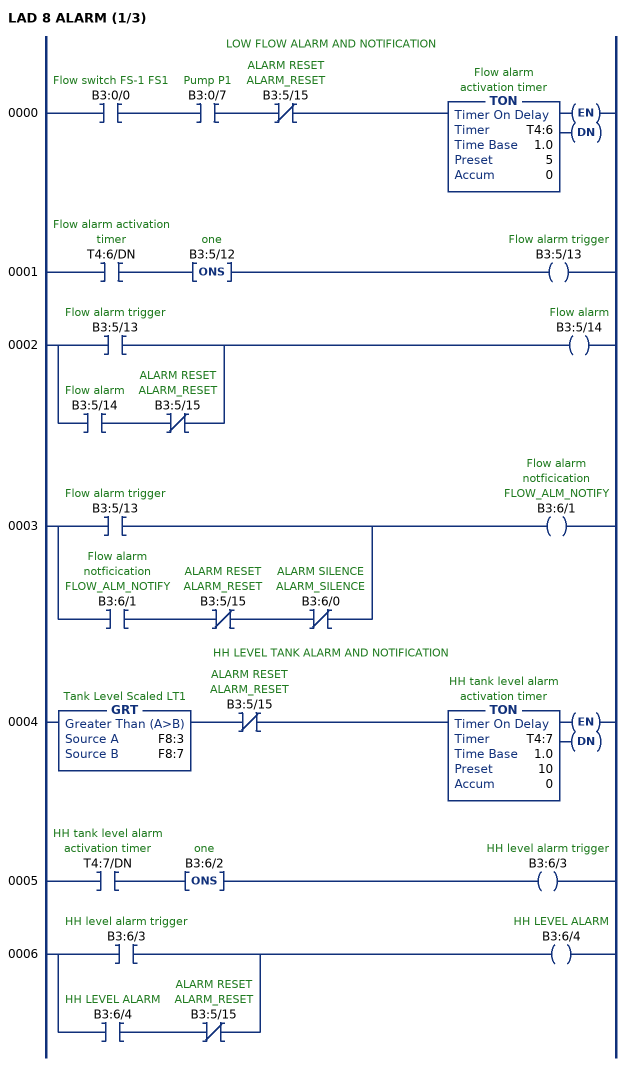
% Rung: 0 %
% LOW FLOW ALARM AND NOTIFICATION %
SOR XIC B3:0/0 XIC B3:0/7 XIO B3:5/15 TON T4:6 1.0 5 0 EOR
%   B3:0/0  FS1  "Flow switch FS-1" %
%   B3:0/7  P1  "Pump" %
%   B3:5/15  ALARM_RESET  "ALARM RESET" %
%   T4:6  "Flow alarm activation timer" %
% Rung: 1 %
SOR XIC T4:6/DN ONS B3:5/12 OTE B3:5/13 EOR
%   T4:6  "Flow alarm activation timer" %
%   B3:5/12  "one" %
%   B3:5/13  "Flow alarm trigger" %
% Rung: 2 %
SOR BST XIC B3:5/13 NXB XIC B3:5/14 XIO B3:5/15 BND OTE B3:5/14 EOR
%   B3:5/13  "Flow alarm trigger" %
%   B3:5/14  "Flow alarm" %
%   B3:5/15  ALARM_RESET  "ALARM RESET" %
% Rung: 3 %
SOR BST XIC B3:5/13 NXB XIC B3:6/1 XIO B3:5/15 XIO B3:6/0 BND OTE B3:6/1 EOR
%   B3:5/13  "Flow alarm trigger" %
%   B3:6/1  FLOW_ALM_NOTIFY  "Flow alarm notficication" %
%   B3:5/15  ALARM_RESET  "ALARM RESET" %
%   B3:6/0  ALARM_SILENCE  "ALARM SILENCE" %
% Rung: 4 %
% HH LEVEL TANK ALARM AND NOTIFICATION %
SOR GRT F8:3 F8:7 XIO B3:5/15 TON T4:7 1.0 10 0 EOR
%   F8:3  LT1  "Tank Level Scaled" %
%   F8:7  HH_LEVEL_SP  "HH Tank level (set on the HMI)" %
%   B3:5/15  ALARM_RESET  "ALARM RESET" %
%   T4:7  "HH tank level alarm activation timer" %
% Rung: 5 %
SOR XIC T4:7/DN ONS B3:6/2 OTE B3:6/3 EOR
%   T4:7  "HH tank level alarm activation timer" %
%   B3:6/2  "one" %
%   B3:6/3  "HH level alarm trigger" %
% Rung: 6 %
SOR BST XIC B3:6/3 NXB XIC B3:6/4 XIO B3:5/15 BND OTE B3:6/4 EOR
%   B3:6/3  "HH level alarm trigger" %
%   B3:6/4  "HH LEVEL ALARM" %
%   B3:5/15  ALARM_RESET  "ALARM RESET" %

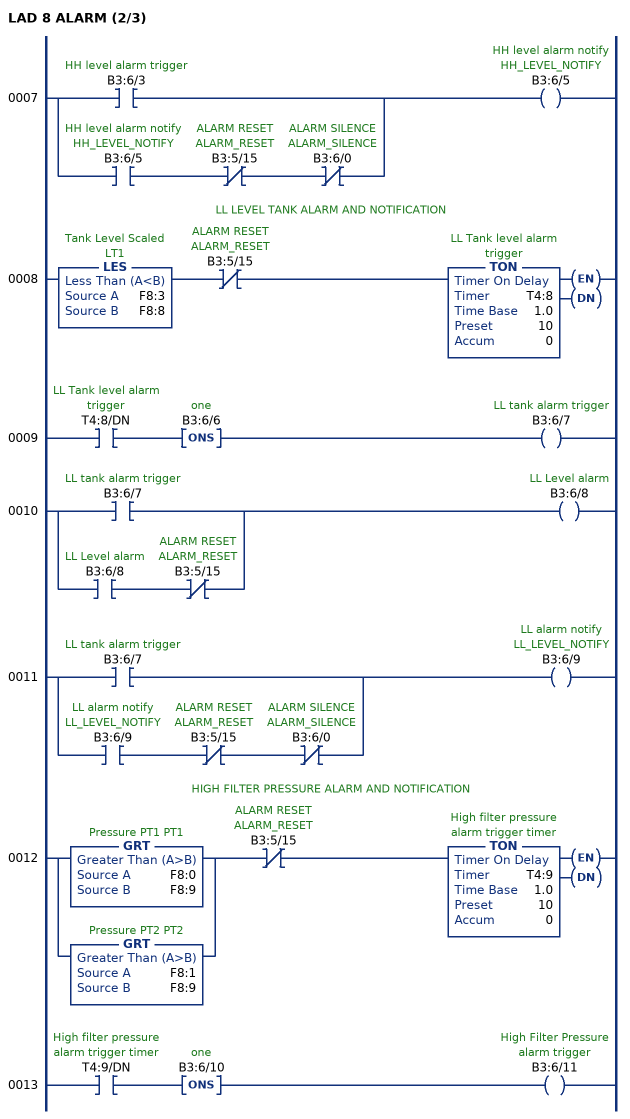
% Rung: 7 %
SOR BST XIC B3:6/3 NXB XIC B3:6/5 XIO B3:5/15 XIO B3:6/0 BND OTE B3:6/5 EOR
%   B3:6/3  "HH level alarm trigger" %
%   B3:6/5  HH_LEVEL_NOTIFY  "HH level alarm notify" %
%   B3:5/15  ALARM_RESET  "ALARM RESET" %
%   B3:6/0  ALARM_SILENCE  "ALARM SILENCE" %
% Rung: 8 %
% LL LEVEL TANK ALARM AND NOTIFICATION %
SOR LES F8:3 F8:8 XIO B3:5/15 TON T4:8 1.0 10 0 EOR
%   F8:3  LT1  "Tank Level Scaled" %
%   F8:8  LL_LEVEL_SP  "LL level (set from HMI)" %
%   B3:5/15  ALARM_RESET  "ALARM RESET" %
%   T4:8  "LL Tank level alarm trigger" %
% Rung: 9 %
SOR XIC T4:8/DN ONS B3:6/6 OTE B3:6/7 EOR
%   T4:8  "LL Tank level alarm trigger" %
%   B3:6/6  "one" %
%   B3:6/7  "LL tank alarm trigger" %
% Rung: 10 %
SOR BST XIC B3:6/7 NXB XIC B3:6/8 XIO B3:5/15 BND OTE B3:6/8 EOR
%   B3:6/7  "LL tank alarm trigger" %
%   B3:6/8  "LL Level alarm" %
%   B3:5/15  ALARM_RESET  "ALARM RESET" %
% Rung: 11 %
SOR BST XIC B3:6/7 NXB XIC B3:6/9 XIO B3:5/15 XIO B3:6/0 BND OTE B3:6/9 EOR
%   B3:6/7  "LL tank alarm trigger" %
%   B3:6/9  LL_LEVEL_NOTIFY  "LL alarm notify" %
%   B3:5/15  ALARM_RESET  "ALARM RESET" %
%   B3:6/0  ALARM_SILENCE  "ALARM SILENCE" %
% Rung: 12 %
% HIGH FILTER PRESSURE ALARM AND NOTIFICATION %
SOR BST GRT F8:0 F8:9 NXB GRT F8:1 F8:9 BND XIO B3:5/15 TON T4:9 1.0 10 0 EOR
%   F8:0  PT1  "Pressure PT1" %
%   F8:9  H_PRES_SP  "High pressure (set from HMI)" %
%   F8:1  PT2  "Pressure PT2" %
%   B3:5/15  ALARM_RESET  "ALARM RESET" %
%   T4:9  "High filter pressure alarm trigger timer" %
% Rung: 13 %
SOR XIC T4:9/DN ONS B3:6/10 OTE B3:6/11 EOR
%   T4:9  "High filter pressure alarm trigger timer" %
%   B3:6/10  "one" %
%   B3:6/11  "High Filter Pressure alarm trigger" %

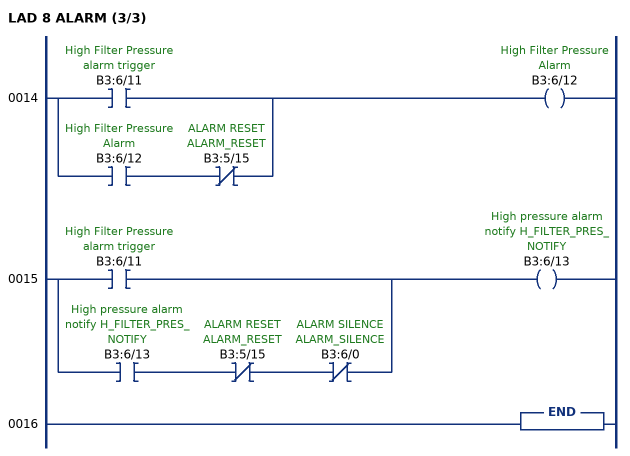
% Rung: 14 %
SOR BST XIC B3:6/11 NXB XIC B3:6/12 XIO B3:5/15 BND OTE B3:6/12 EOR
%   B3:6/11  "High Filter Pressure alarm trigger" %
%   B3:6/12  "High Filter Pressure Alarm" %
%   B3:5/15  ALARM_RESET  "ALARM RESET" %
% Rung: 15 %
SOR BST XIC B3:6/11 NXB XIC B3:6/13 XIO B3:5/15 XIO B3:6/0 BND OTE B3:6/13 EOR
%   B3:6/11  "High Filter Pressure alarm trigger" %
%   B3:6/13  H_FILTER_PRES_NOTIFY  "High pressure alarm notify" %
%   B3:5/15  ALARM_RESET  "ALARM RESET" %
%   B3:6/0  ALARM_SILENCE  "ALARM SILENCE" %
% Rung: 16 %
SOR END EOR

LADDER 9 "SIMULATION"    % SIMULATED IO %
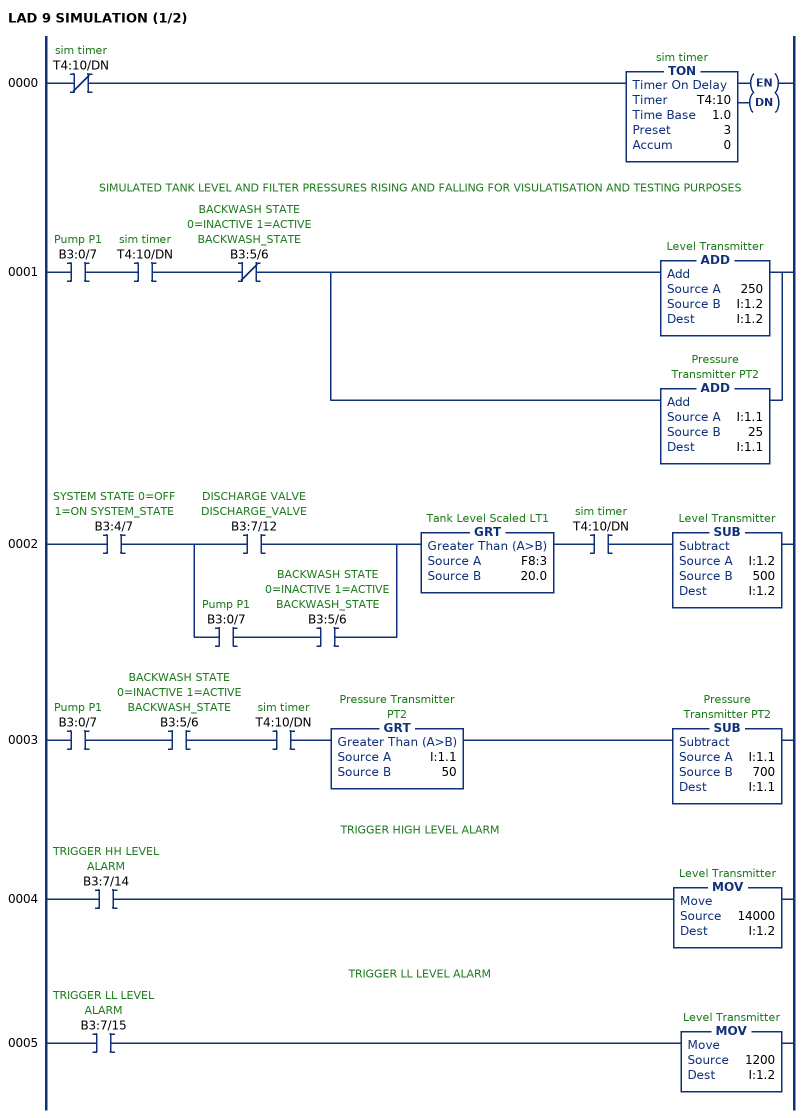
% Rung: 0 %
SOR XIO T4:10/DN TON T4:10 1.0 3 0 EOR
%   T4:10  "sim timer" %
% Rung: 1 %
% SIMULATED TANK LEVEL AND FILTER PRESSURES RISING AND FALLING FOR VISULATISATION AND TESTING PURPOSES %
SOR XIC B3:0/7 XIC T4:10/DN XIO B3:5/6 BST ADD 250 I:1.2 I:1.2 NXB ADD I:1.1 25 I:1.1 BND EOR
%   B3:0/7  P1  "Pump" %
%   T4:10  "sim timer" %
%   B3:5/6  BACKWASH_STATE  "BACKWASH STATE 0=INACTIVE 1=ACTIVE" %
%   I:1.2  "Level Transmitter" %
%   I:1.1  "Pressure Transmitter PT2" %
% Rung: 2 %
SOR XIC B3:4/7 BST XIC B3:7/12 NXB XIC B3:0/7 XIC B3:5/6 BND GRT F8:3 20.0 XIC T4:10/DN SUB I:1.2 500 I:1.2 EOR
%   B3:4/7  SYSTEM_STATE  "SYSTEM STATE 0=OFF 1=ON" %
%   B3:7/12  DISCHARGE_VALVE  "DISCHARGE VALVE" %
%   B3:0/7  P1  "Pump" %
%   B3:5/6  BACKWASH_STATE  "BACKWASH STATE 0=INACTIVE 1=ACTIVE" %
%   F8:3  LT1  "Tank Level Scaled" %
%   T4:10  "sim timer" %
%   I:1.2  "Level Transmitter" %
% Rung: 3 %
SOR XIC B3:0/7 XIC B3:5/6 XIC T4:10/DN GRT I:1.1 50 SUB I:1.1 700 I:1.1 EOR
%   B3:0/7  P1  "Pump" %
%   B3:5/6  BACKWASH_STATE  "BACKWASH STATE 0=INACTIVE 1=ACTIVE" %
%   T4:10  "sim timer" %
%   I:1.1  "Pressure Transmitter PT2" %
% Rung: 4 %
% TRIGGER HIGH LEVEL ALARM %
SOR XIC B3:7/14 MOV 14000 I:1.2 EOR
%   B3:7/14  "TRIGGER HH LEVEL ALARM" %
%   I:1.2  "Level Transmitter" %
% Rung: 5 %
% TRIGGER LL LEVEL ALARM %
SOR XIC B3:7/15 MOV 1200 I:1.2 EOR
%   B3:7/15  "TRIGGER LL LEVEL ALARM" %
%   I:1.2  "Level Transmitter" %

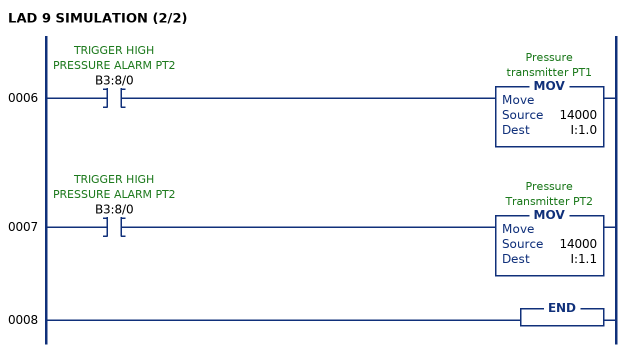
% Rung: 6 %
SOR XIC B3:8/0 MOV 14000 I:1.0 EOR
%   B3:8/0  "TRIGGER HIGH PRESSURE ALARM PT2" %
%   I:1.0  "Pressure transmitter PT1" %
% Rung: 7 %
SOR XIC B3:8/0 MOV 14000 I:1.1 EOR
%   B3:8/0  "TRIGGER HIGH PRESSURE ALARM PT2" %
%   I:1.1  "Pressure Transmitter PT2" %
% Rung: 8 %
SOR END EOR

LADDER 10 "SETTOAUTO"
